// TIA Portal V18 export
DATA_BLOCK "vessel_1"   // DB81
{ S7_Optimized_Access := 'TRUE' }
VERSION : 0.1
// stored: AutoNumber true, DBAccessibleFromOPCUA true, IsOnlyStoredInLoadMemory false, IsRetainMemResEnabled false, IsWriteProtectedInAS false, MemoryReserve 100
   VAR RETAIN
      "Duration pressure equalization" : Struct
         "A" : Int;
         "B" : Int;
      END_STRUCT;
      "amibient pressure" : Int;
      "hysteresis ambient pressure" : Int;
      "working pressure" : Struct
         "A" : Real;
         "A+" : Real;
         "A-" : Real;
         "B" : Real;
         "B+" : Real;
         "B-" : Real;
      END_STRUCT;
      "working pressure hysteresis" : Struct
         "A" : Real;
         "B" : Real;
      END_STRUCT;
   END_VAR
   VAR
      "Vaccum sensor selection" : Struct
         "selection A" : Int;
         "selection B" : Int;
         "A selected" : Bool;
         "B selected" : Bool;
         "A or B selected" : Bool;
      END_STRUCT;
      "Ready status" : Struct
         A1 : Int;
         A2 : Int;
         B1 : Int;
      END_STRUCT;
      "Evacuation set Vaccum" : Struct
         A1 : Int;
         A2 : Int;
         B1 : Int;
      END_STRUCT;
      "Evacuation Real vaccum" : Struct
         A1 : Int;
         A2 : Int;
         B1 : Int;
      END_STRUCT;
      "Evacuation Time set" : Struct
         A1 : Int;
         A2 : Int;
         B1 : Int;
      END_STRUCT;
      "Evacuation Time Real" : Struct
         A1 : Int;
         A2 : Int;
         B1 : Int;
      END_STRUCT;
   END_VAR
   VAR RETAIN
      "Active vessel" : Struct
         A1 : Bool;
         A2 : Bool;
         "A" : Bool;
         B1 : Bool;
      END_STRUCT;
      "preparation status" : Struct
         A1 : Int;
         A2 : Int;
         B1 : Int;
      END_STRUCT;
      "monitor status" : Struct
         "A" : Int;
         "B" : Int;
         C : Int;
      END_STRUCT;
      "Activate vessel" : Struct
         A1 : Bool;
         A2 : Bool;
         B1 : Bool;
      END_STRUCT;
   END_VAR
   VAR
      Ready : Struct
         A1 : Bool;
         A2 : Bool;
         B1 : Bool;
      END_STRUCT;
      "Activate vessel HMI" : Struct
         A1 : Bool;
         A2 : Bool;
         B1 : Bool;
      END_STRUCT;
      "DeActivate vessel HMI" : Struct
         A1 : Bool;
         A2 : Bool;
         B1 : Bool;
      END_STRUCT;
   END_VAR
BEGIN
END_DATA_BLOCK
